{attribute 'GeneratedUsingTerminal: EL2595-0000-0018'}
{attribute addProperty BoxType "EL2595-0000-0018"}
{attribute addProperty Id "EtcSlaveTerminalBaseDOX_StatusAT %I*DOX_Status_AED8A12A6DOX_ControlAT %Q*DOX_Control_75D5C9E23WcStateAT %I*WcState_9091E0EB2InfoDataAT %I*InfoData_32EB74EA10"}
{attribute addProperty CRC "3537663653"}
{attribute addProperty Size "21"}
TYPE EL2595_D2DC76A5 EXTENDS EtcSlaveTerminalBase :
STRUCT
	{attribute addProperty Name "DOX_Status"}
	DOX_Status : DOX_Status_AED8A12A;
	{attribute addProperty Name "DOX_Control"}
	DOX_Control : DOX_Control_75D5C9E2;
	{attribute addProperty Name "WcState"}
	WcState : WcState_9091E0EB;
	{attribute addProperty Name "InfoData"}
	InfoData : InfoData_32EB74EA;
END_STRUCT
END_TYPE

(* stored: Version 1.2.0.0, ProductVersion 3.1.4024.9
   DUT EL2595_D2DC76A5: Id {6e5a4661-40aa-4bff-9066-77fd3d5cf1f5} *)
